// Block: A0301_Ribaltatore_PERS

DATA_BLOCK A0301_Ribaltatore_PERS
VERSION : 0.1
   NON_RETAIN
   VAR
      Par_Manu : Positioning_EPOS_Machine_Par;
      Par_Aut : A0301_Mach_Ribaltatore_Par;
      Par_Aut_Vel : Struct
         Pos1_Frw : LReal;
         Pos2_Frw : LReal;
         Pos0_Brw : LReal;
      END_STRUCT;
      Pers_Data : Struct
         EncoderAbsolute_Preset_OK : Bool;
         Persistent_ActualPosition : LReal;
      END_STRUCT;
   END_VAR

BEGIN
   // No initialization required
END_DATA_BLOCK
